Universal Robots PolyScope program: _adminCG-PHomeToInvB.urp

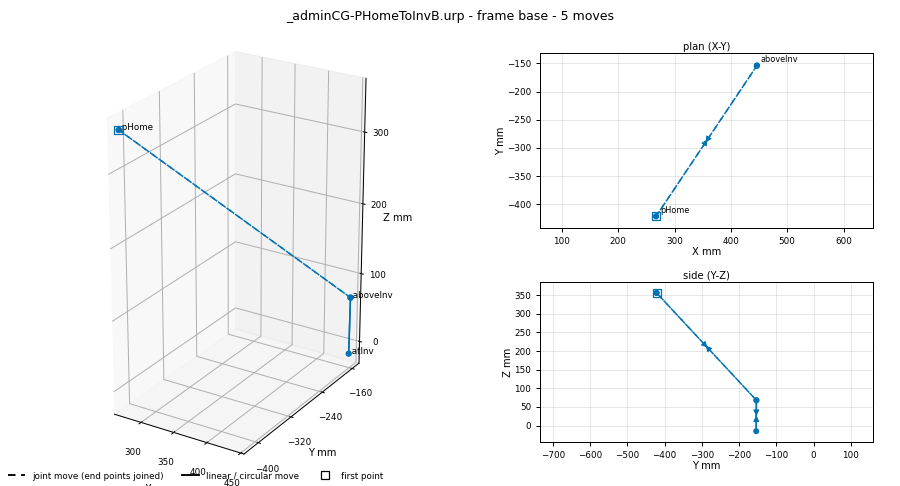
[picture p0: tool path of _adminCG-PHomeToInvB.urp in frame base, 5 of 5 moves have a stored position in this frame; points joined in program order, loops and branches not executed]
Program _adminCG-PHomeToInvB (installation=admin directory=/programs/THU_530PM createdIn=3.8.0.61336 lastSavedIn=3.15.8.106339 robotSerialNumber=2015350924)
Calibrated DH parameters: a=[0, -0.425, -0.39225, 0, 0, 0]; d=[0.089159, 0, 0, 0.10915, 0.09465, 0.0823]; alpha=[1.570796, 0, 0, 1.570796, -1.570796, 0]; deltaTheta=[0, 0, 0, 0, 0, 0]
Robot Program (runOnlyOnce=true)
  Set DigitalOutput pin=digital_out[0]; digitalValue=1
  Call _adminLinearIndex2
  MoveJ speed 60 deg/s, acceleration 80 deg/s^2 (useActiveTCP=true)
    Waypoint pHome: TCP in base x=267.077 y=-421.526 z=355.862 mm, rx=1.114 ry=1.1061 rz=0.0051 rad; joints [-45.007, -90.005, -89.993, -90.005, 90, -0.004] deg; flange x=267.08 y=-421.53 z=431.862 mm, rx=1.2021 ry=-2.9025 rz=-0.0001 rad
    Waypoint aboveInv: TCP in base x=446.318 y=-153.704 z=67.867 mm, rx=1.1163 ry=1.1066 rz=-0.0014 rad; joints [-5.61, -102.047, -123.143, -45.023, 89.931, 39.674] deg; flange x=446.609 y=-153.641 z=143.867 mm, rx=1.1936 ry=-2.9019 rz=-0.0011 rad
  MoveL speed 250 mm/s, acceleration 1200 mm/s^2 (useActiveTCP=true) feature=Base
    Waypoint atInv: TCP in base x=445.782 y=-154.212 z=-15.17 mm, rx=1.1163 ry=1.1067 rz=-0.0013 rad; joints [-5.68, -112.814, -126.528, -30.875, 89.932, 39.602] deg; flange x=446.077 y=-154.151 z=60.829 mm, rx=1.1936 ry=-2.9018 rz=-0.0012 rad
    Set DigitalOutput pin=digital_out[0]; digitalValue=0
    Wait Sleep waitTime=1
    Waypoint aboveInv: TCP in base x=446.318 y=-153.704 z=67.867 mm, rx=1.1163 ry=1.1066 rz=-0.0014 rad; joints [-5.61, -102.047, -123.143, -45.023, 89.931, 39.674] deg; flange x=446.609 y=-153.641 z=143.867 mm, rx=1.1936 ry=-2.9019 rz=-0.0011 rad
  MoveJ speed 180 deg/s, acceleration 100 deg/s^2 (useActiveTCP=true)
    Waypoint phome: TCP in base x=267.106 y=-421.453 z=355.828 mm, rx=1.114 ry=1.1062 rz=0.0052 rad; joints [-45, -90.001, -90.002, -90.005, 90.003, -0.002] deg; flange x=267.11 y=-421.463 z=431.828 mm, rx=1.2023 ry=-2.9024 rz=-0.0002 rad
SubProgram -> _adminLinearIndex2
SubProgram _adminLinearIndex2 (keepSynchronizedWithDisk=false) programFile=/programs/me345_admin/_adminLinearIndex2.urp
  Folder Move_linear_slide_Index2
    var_1 := False
    Loop While (checkContinuously=false) expression=var_1≟ False
      var_1 := socket_open("10.241.34.52",4001)
    var_3 := 1
    Send := "s r0x24 21"
    Script: socket_send_string(Send)
    Script: socket_send_byte(13)
    Send_Reply := socket_read_string()
    Send := "s r0xca 56389"
    Script: socket_send_string(Send)
    Script: socket_send_byte(13)
    Send_Reply := socket_read_string()
    Send := "t 1"
    Script: socket_send_string(Send)
    Script: socket_send_byte(13)
    Send_Reply := socket_read_string()
    Loop While (checkContinuously=false) expression=var_3≠0
      Send := "g r0xA0"
      Script: socket_send_string(Send)
      Script: socket_send_byte(13)
      var_3 := socket_get_var("v")
      Wait Sleep waitTime=0.1
    Script: socket_close()
    Script: sync()
